# EPICS autosave request: stdApp/Db/userCalcN_settings.req
# FILE... userCalcN_settings.req
# USAGE.. userCalcN.db fields autosave'd.

file swait_settings.req P=$(P)userCalc$(N)
